Staubli VAL3: SingleMove.pgx

public program SingleMove(num x_nType, jointRx x_j, pointRx x_pM, pointRx x_pE, tool x_tTool, mdesc x_m, trsf x_trExtAxis)
  local pointRx l_pP[2]
begin
  if x_nType<1 or x_nType>3
    return
  endIf

  resize(nAxesData,1,nAxesSum)
  nAxesData[0]=x_trExtAxis.x
  if nAxesSum>=2
    nAxesData[1]=x_trExtAxis.y

  endIf



  if !bMoveType or x_nType==1

    switch x_nType
      case 1
        $Xmovej(x_j,nAxesData,x_tTool,x_m)
      break


      case 2
        $Xmovel(x_pE,nAxesData,x_tTool,x_m)
      break

      case 3
        $Xmovec(x_pM,x_pE,nAxesData,x_tTool,x_m)
      break


    endSwitch
    return


  endIf





  //2014.12.04
  //对于离线进行修改
  //fFrame.trsf={0,0,0,0,0,0}
  if bMoveType
    $XframeLink(fFrame)
  else
    link(fFrame,world)
  endIf





  link(l_pP[0],fFrame)
  link(l_pP[1],fFrame)


  l_pP[0].trsf=x_pM.trsf
  l_pP[1].trsf=x_pE.trsf

  //×××××××××××××××××××××××××××××××××××××××××××
  switch x_nType
    case 1
      $Xmovej(x_j,nAxesData,x_tTool,x_m)
    break

    case 2
      $Xmovel(l_pP[1],nAxesData,x_tTool,x_m)
    break

    case 3
      $Xmovec(l_pP[0],l_pP[1],nAxesData,x_tTool,x_m)
    break

  endSwitch


end
